(* CoDeSys 2.3 export: F_READ_SENSOR_KG.EXP *)

(* POU FUN/PARAMETERS/F_READ_SENSOR_KG, ST *)
FUNCTION F_READ_SENSOR_KG : BOOL
VAR_INPUT
END_VAR
VAR_IN_OUT
	stSensor : ST_SENSOR_KG;
	fbIdList : FB_IDLIST;
END_VAR
VAR
END_VAR
stSensor.Cal_K := F_IDLIST_GETREAL( CONCAT(stSensor.Name, '_K' ), fbIdList );
stSensor.Cal_C := F_IDLIST_GETREAL( CONCAT(stSensor.Name, '_C' ), fbIdList );
END_FUNCTION
